FUNCTION_BLOCK FB_Setter

VAR_INPUT			// Input Variables
	dMotorState  : BOOL;
	dMotorSpeed  : INT;
	dFV1_Percent : INT;
	dLV1_Percent : INT;
	dLV2_Percent : INT;
	dLV3_Percent : INT;
END_VAR

(*VAR_IN_OUT			// Pass by Reference
	MotorState  : BOOL;
	MotorSpeed  : INT;
	FV1_Percent : INT;
	LV1_Percent : INT;
	LV2_Percent : INT;
	LV3_Percent : INT;
END_VAR*)

(*	// Send input to output
MotorState  := dMotorState;
MotorSpeed  := dMotorSpeed;
FV1_Percent := dFV1_Percent;
LV1_Percent := dLV1_Percent;
LV2_Percent := dLV2_Percent;
LV3_Percent := dLV3_Percent;*)

END_FUNCTION_BLOCK

(* stored: Version 1.1.0.1, ProductVersion 3.1.4024.12
   POU FB_Setter: Id {26f2809c-62d5-41d8-852e-0b01ce281a8d}, SpecialFunc None *)
